FUNCTION_BLOCK FB_FieldCodecEnum EXTENDS FB_FieldCodec
VAR_INPUT
END_VAR
VAR_OUTPUT
END_VAR
VAR
    nValue : DINT;
END_VAR

METHOD CalculatePackedDataSize : HRESULT
VAR_INPUT CONSTANT
	anyFirstElem	: T_Any;
	nLength	        : UDINT;
END_VAR
VAR_OUTPUT
    nPackedDataSize : UDINT;
END_VAR
VAR
    anyItem : T_Any;
    i : UDINT;
    nCopySize : UDINT;
    nTmp : DINT;
    retVal : UDINT;
END_VAR
nPackedDataSize := 0;

IF anyFirstElem.pValue = NULL OR anyFirstElem.TypeClass <> __SYSTEM.TYPE_CLASS.TYPE_ENUM THEN
    CalculatePackedDataSize := E_HRESULTAdsErr.INVALIDDATA;
    RETURN;
END_IF

nCopySize := MIN(TO_UDINT(anyFirstElem.diSize), SIZEOF(nTmp));
IF nCopySize = 0 THEN
    CalculatePackedDataSize := E_HRESULTAdsErr.INVALIDDATA;
    RETURN;
END_IF

IF nLength < 1 THEN
    CalculatePackedDataSize := S_OK;
    RETURN;
END_IF

anyItem := anyFirstElem;

FOR i := 0 TO nLength - 1 DO
    anyItem.pValue := anyFirstElem.pValue + (i * TO_UDINT(anyFirstElem.diSize));
    nTmp := 0;
    retVal := MEMCPY(destAddr:= ADR(nTmp), srcAddr:= anyItem.pValue, n:= nCopySize);
    IF retVal = 0 THEN
        CalculatePackedDataSize := E_HRESULTAdsErr.INVALIDDATA;
        RETURN;
    END_IF
    nPackedDataSize := nPackedDataSize + F_ComputeInt32Size(nTmp);
END_FOR

CalculatePackedDataSize := S_OK;
END_METHOD

METHOD IsPackedRepeatedField : BOOL
VAR_INPUT
	nTag	: UDINT;
END_VAR
IsPackedRepeatedField := F_IsPackedRepeatedField(nTag);
END_METHOD


METHOD ValueReader : HRESULT
VAR_IN_OUT
    stCtx : ST_ParseContext;
END_VAR
VAR_OUTPUT
	anyOut	: T_Any;
END_VAR
nValue := 0;
ValueReader := F_ParseRawVarint32(stCtx, nValue);
IF FAILED(ValueReader) THEN
    RETURN;
END_IF

anyOut := F_ToAnyType(anyArg:= nValue);
END_METHOD

METHOD ValueWriter : HRESULT
VAR_IN_OUT
    stCtx  : ST_WriteContext;
END_VAR
VAR_INPUT
	anyIn	: T_ANY;
END_VAR
VAR
    nCopySize : UDINT;
    retVal : UDINT;
END_VAR
IF anyIn.pValue = NULL OR anyIn.TypeClass <> __SYSTEM.TYPE_CLASS.TYPE_ENUM THEN
    ValueWriter := E_HRESULTAdsErr.INVALIDDATA;
    RETURN;
END_IF

nCopySize := MIN(TO_UDINT(anyIn.diSize), SIZEOF(nValue));
IF nCopySize = 0 THEN
    ValueWriter := E_HRESULTAdsErr.INVALIDDATA;
    RETURN;
END_IF

nValue := 0;
retVal := MEMCPY(destAddr:= ADR(nValue), srcAddr:= anyIn.pValue, n:= nCopySize);
IF retVal = 0 THEN
    ValueWriter := E_HRESULTAdsErr.INVALIDDATA;
    RETURN;
END_IF

ValueWriter := F_WriteEnum(stCtx, nValue);
END_METHOD

END_FUNCTION_BLOCK

(* stored: Version 1.1.0.1
   POU FB_FieldCodecEnum: Id {10e15aa8-0b38-41f2-b906-d6a58244fe65}, SpecialFunc None
   Method CalculatePackedDataSize: Id {84002809-9a36-4d76-bc25-8546d7cb8423}
   Method IsPackedRepeatedField: Id {9f999de1-21ca-4b25-b85b-9904dba50910}
   Method ValueReader: Id {0e32fa9a-f796-4486-8d6e-ecaa09bc162c}
   Method ValueWriter: Id {fe225455-b643-4ce0-90f6-4406fc4cfd97} *)
